FUNCTION_BLOCK Plant
  (* Standard: 61499-2 *)
  (* Version 0,1, 2015-00-15, Th?o, PC_THEO *)
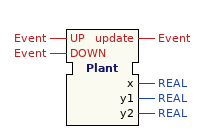
  EVENT_INPUT
    UP;
    DOWN;
  END_EVENT
  EVENT_OUTPUT
    update;
  END_EVENT
  VAR_OUTPUT
    x : REAL;
    y1 : REAL;
    y2 : REAL;
  END_VAR
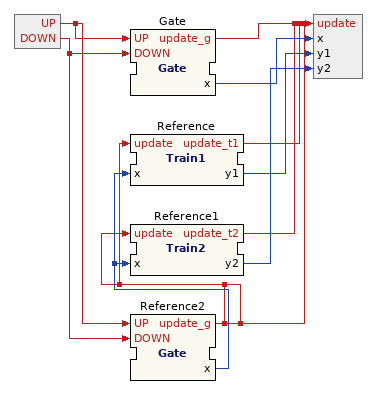
  FBS
    Gate : Gate;
    Reference : Train1;
    Reference1 : Train2;
    Reference2 : Gate;
  END_FBS
  EVENT_CONNECTIONS
    UP TO Gate.UP;
    UP TO Reference2.UP;
    DOWN TO Gate.DOWN;
    DOWN TO Reference2.DOWN;
    Gate.update_g TO update;
    Reference.update_t1 TO update;
    Reference1.update_t2 TO update;
    Reference2.update_g TO update;
    Reference2.update_g TO Reference1.update;
    Reference2.update_g TO Reference.update;
  END_CONNECTIONS
  DATA_CONNECTIONS
    Gate.x TO x;
    Reference.y1 TO y1;
    Reference1.y2 TO y2;
    Reference2.x TO Reference.x;
    Reference2.x TO Reference1.x;
  END_CONNECTIONS
END_FUNCTION_BLOCK
